TYPE E_PositioningState :
(
	INIT,
	STANDBY,
	POSITIONING_ABSOLUTE,
	STOPPING,
	HALTING,
	POSITIONING_FINISHED,
	MANUAL_MODE,
	COMMISSIONING,
	ERROR
);
END_TYPE

(* stored: Version 1.1.0.1, ProductVersion 3.1.4024.9
   DUT E_PositioningState: Id {69ca3900-ce23-4e0c-8fac-f41131a07d73} *)
